FUNCTION_BLOCK ArraySquared (* Basic FB with empty ECC *)
  (* Standard: 61499-2 *)
  (* Version 1.0, 2020-07-23, Candra Wardaya, UGM *)
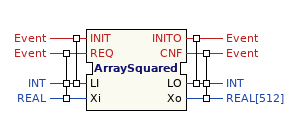
  EVENT_INPUT
    INIT WITH LI; (* Initialization Input *)
    REQ WITH LI, Xi; (* Execution Request *)
  END_EVENT
  EVENT_OUTPUT
    INITO WITH LO; (* Initialization Output *)
    CNF WITH LO, Xo; (* Confirmation of Execution *)
  END_EVENT
  VAR_INPUT
    LI : INT; (* Array Length Input *)
    Xi : REAL; (* Single Real Input *)
  END_VAR
  VAR_OUTPUT
    LO : INT; (* Array Length Output *)
    Xo : ARRAY [0..511] OF REAL; (* Array Real Squared Output *)
  END_VAR
  VAR
    L : INT; (* Internal Variable *)
    i : INT; (* Internal Variable *)
  END_VAR
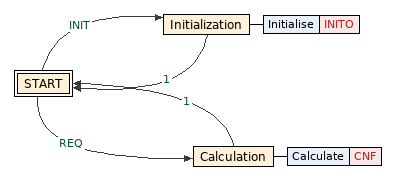
  EC_STATES
    START; (* Initial State *)
    Initialization : Initialise -> INITO;
    Calculation : Calculate -> CNF;
  END_STATES
  EC_TRANSITIONS
    START TO Initialization := INIT;
    Initialization TO START := 1;
    START TO Calculation := REQ;
    Calculation TO START := 1;
  END_TRANSITIONS
  ALGORITHM Initialise IN ST: (* New Algorithm *)

  END_ALGORITHM
  ALGORITHM Calculate IN ST: (* New Algorithm *)
L := LI;

for i := 1 to L-1 do
	Xo[i-1] := Xo[i];
end_for;

Xo[L-1] := Xi*Xi;

LO := L;
  END_ALGORITHM
END_FUNCTION_BLOCK
